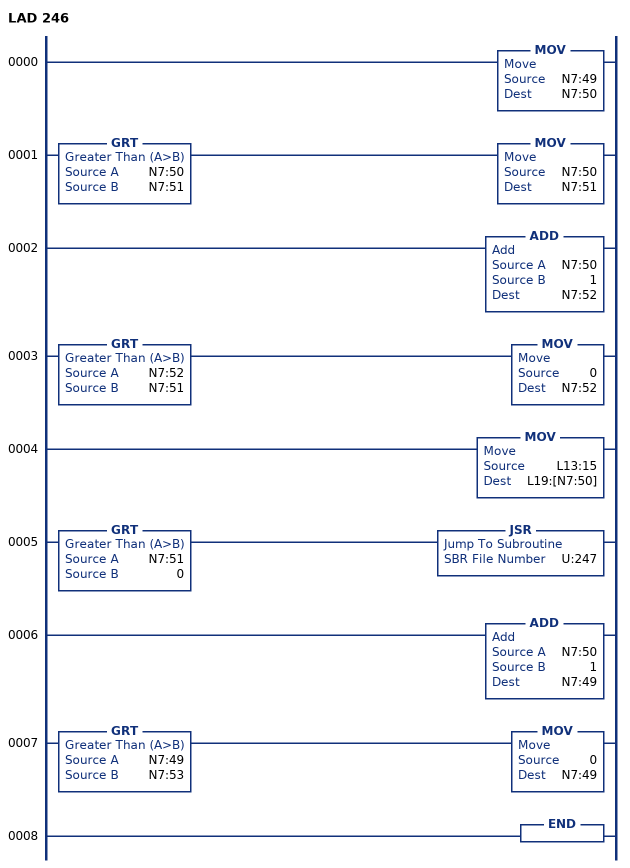
% Rung: 0 %
SOR MOV N7:49 N7:50 EOR
% Rung: 1 %
SOR GRT N7:50 N7:51 MOV N7:50 N7:51 EOR
% Rung: 2 %
SOR ADD N7:50 1 N7:52 EOR
% Rung: 3 %
SOR GRT N7:52 N7:51 MOV 0 N7:52 EOR
% Rung: 4 %
SOR MOV L13:15 L19:[N7:50] EOR
% Rung: 5 %
SOR GRT N7:51 0 JSR U:247 EOR
% Rung: 6 %
SOR ADD N7:50 1 N7:49 EOR
% Rung: 7 %
SOR GRT N7:49 N7:53 MOV 0 N7:49 EOR
% Rung: 8 %
SOR END EOR

LADDER 247
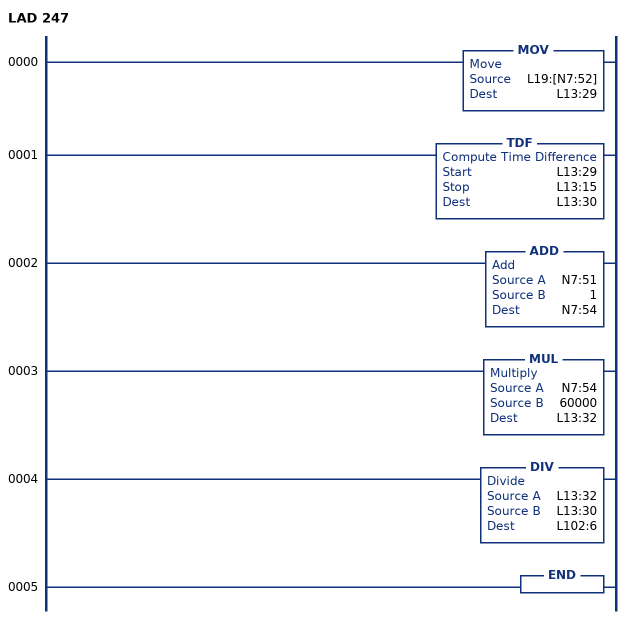
% Rung: 0 %
SOR MOV L19:[N7:52] L13:29 EOR
% Rung: 1 %
SOR TDF L13:29 L13:15 L13:30 EOR
% Rung: 2 %
SOR ADD N7:51 1 N7:54 EOR
% Rung: 3 %
SOR MUL N7:54 60000 L13:32 EOR
% Rung: 4 %
SOR DIV L13:32 L13:30 L102:6 EOR
% Rung: 5 %
SOR END EOR

LADDER 248
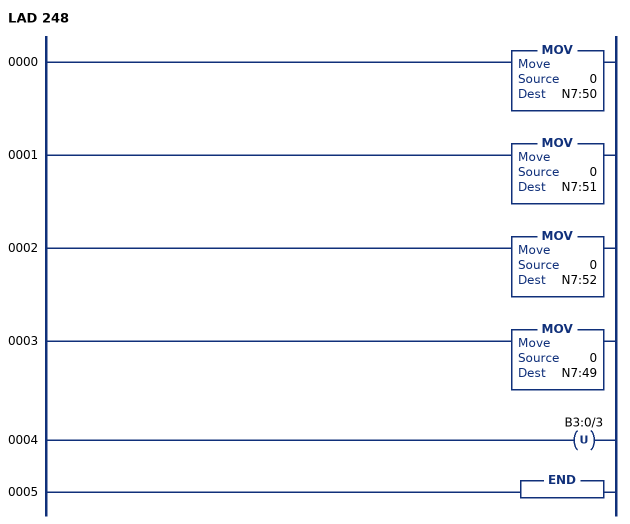
% Rung: 0 %
SOR MOV 0 N7:50 EOR
% Rung: 1 %
SOR MOV 0 N7:51 EOR
% Rung: 2 %
SOR MOV 0 N7:52 EOR
% Rung: 3 %
SOR MOV 0 N7:49 EOR
% Rung: 4 %
SOR OTU B3:0/3 EOR
% Rung: 5 %
SOR END EOR

LADDER 249
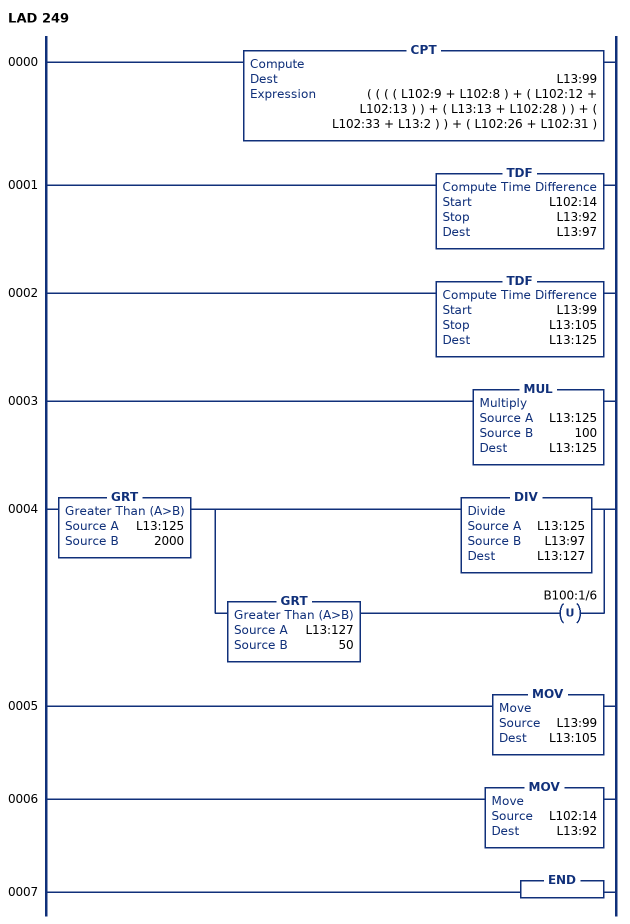
% Rung: 0 %
SOR CPT L13:99 " ( ( ( ( L102:9 + L102:8 ) + ( L102:12 + L102:13 ) ) + ( L13:13 + L102:28 ) ) + ( L102:33 + L13:2 ) ) + ( L102:26 + L102:31 ) " EOR
% Rung: 1 %
SOR TDF L102:14 L13:92 L13:97 EOR
% Rung: 2 %
SOR TDF L13:99 L13:105 L13:125 EOR
% Rung: 3 %
SOR MUL L13:125 100 L13:125 EOR
% Rung: 4 %
SOR GRT L13:125 2000 BST DIV L13:125 L13:97 L13:127 NXB GRT L13:127 50 OTU B100:1/6 BND EOR
% Rung: 5 %
SOR MOV L13:99 L13:105 EOR
% Rung: 6 %
SOR MOV L102:14 L13:92 EOR
% Rung: 7 %
SOR END EOR

LADDER 250
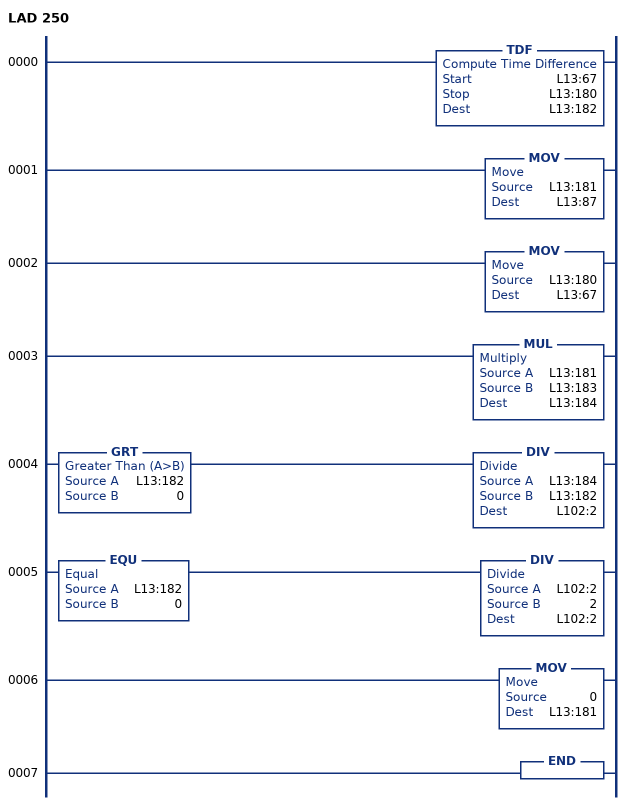
% Rung: 0 %
SOR TDF L13:67 L13:180 L13:182 EOR
% Rung: 1 %
SOR MOV L13:181 L13:87 EOR
% Rung: 2 %
SOR MOV L13:180 L13:67 EOR
% Rung: 3 %
SOR MUL L13:181 L13:183 L13:184 EOR
% Rung: 4 %
SOR GRT L13:182 0 DIV L13:184 L13:182 L102:2 EOR
% Rung: 5 %
SOR EQU L13:182 0 DIV L102:2 2 L102:2 EOR
% Rung: 6 %
SOR MOV 0 L13:181 EOR
% Rung: 7 %
SOR END EOR

LADDER 251
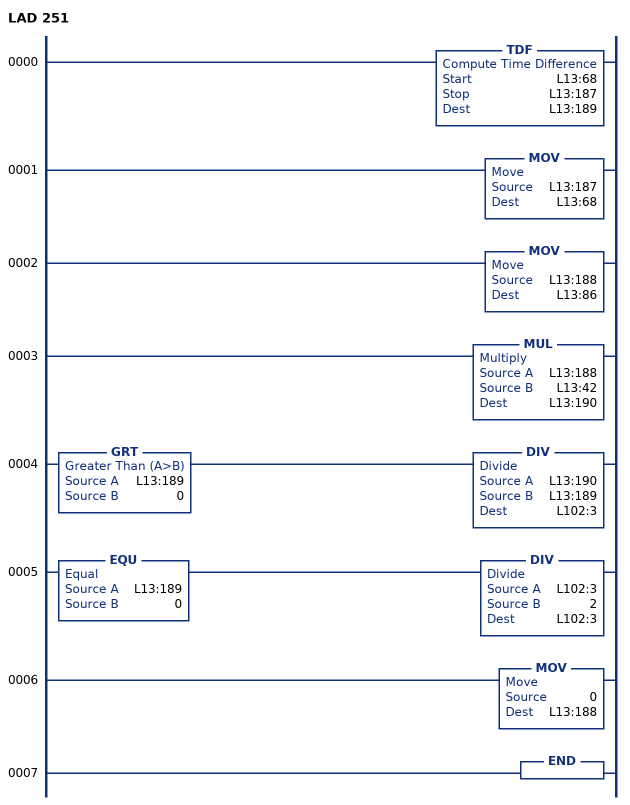
% Rung: 0 %
SOR TDF L13:68 L13:187 L13:189 EOR
% Rung: 1 %
SOR MOV L13:187 L13:68 EOR
% Rung: 2 %
SOR MOV L13:188 L13:86 EOR
% Rung: 3 %
SOR MUL L13:188 L13:42 L13:190 EOR
% Rung: 4 %
SOR GRT L13:189 0 DIV L13:190 L13:189 L102:3 EOR
% Rung: 5 %
SOR EQU L13:189 0 DIV L102:3 2 L102:3 EOR
% Rung: 6 %
SOR MOV 0 L13:188 EOR
% Rung: 7 %
SOR END EOR

LADDER 252
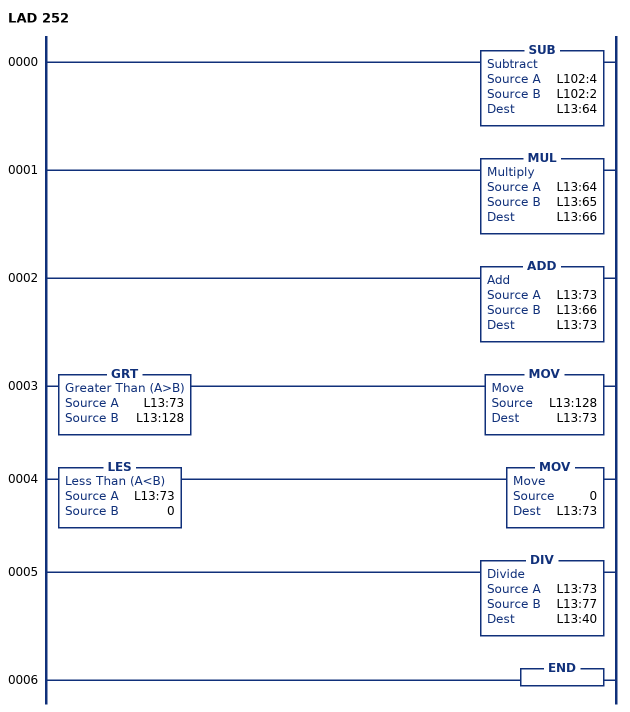
% Rung: 0 %
SOR SUB L102:4 L102:2 L13:64 EOR
% Rung: 1 %
SOR MUL L13:64 L13:65 L13:66 EOR
% Rung: 2 %
SOR ADD L13:73 L13:66 L13:73 EOR
% Rung: 3 %
SOR GRT L13:73 L13:128 MOV L13:128 L13:73 EOR
% Rung: 4 %
SOR LES L13:73 0 MOV 0 L13:73 EOR
% Rung: 5 %
SOR DIV L13:73 L13:77 L13:40 EOR
% Rung: 6 %
SOR END EOR

LADDER 253
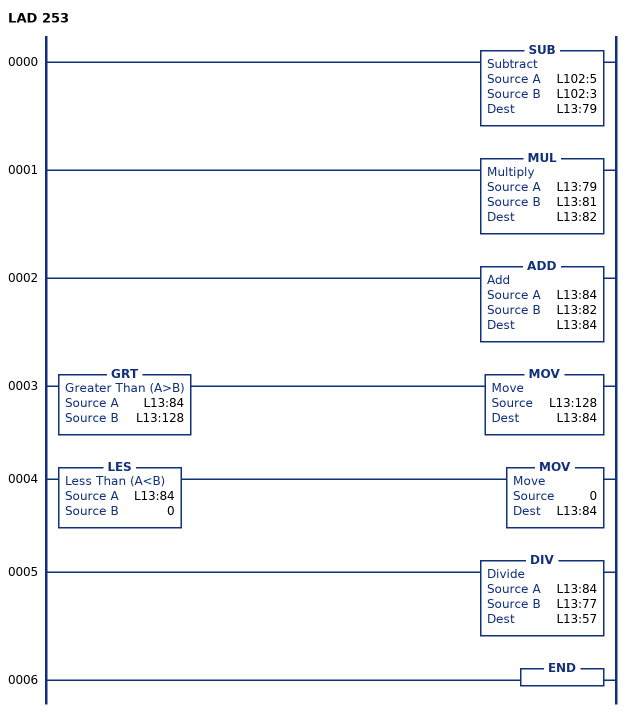
% Rung: 0 %
SOR SUB L102:5 L102:3 L13:79 EOR
% Rung: 1 %
SOR MUL L13:79 L13:81 L13:82 EOR
% Rung: 2 %
SOR ADD L13:84 L13:82 L13:84 EOR
% Rung: 3 %
SOR GRT L13:84 L13:128 MOV L13:128 L13:84 EOR
% Rung: 4 %
SOR LES L13:84 0 MOV 0 L13:84 EOR
% Rung: 5 %
SOR DIV L13:84 L13:77 L13:57 EOR
% Rung: 6 %
SOR END EOR

LADDER 254
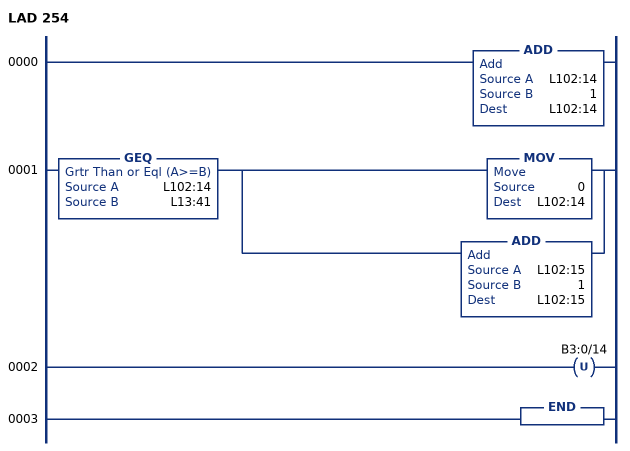
% Rung: 0 %
SOR ADD L102:14 1 L102:14 EOR
% Rung: 1 %
SOR GEQ L102:14 L13:41 BST MOV 0 L102:14 NXB ADD L102:15 1 L102:15 BND EOR
% Rung: 2 %
SOR OTU B3:0/14 EOR
% Rung: 3 %
SOR END EOR

LADDER 255
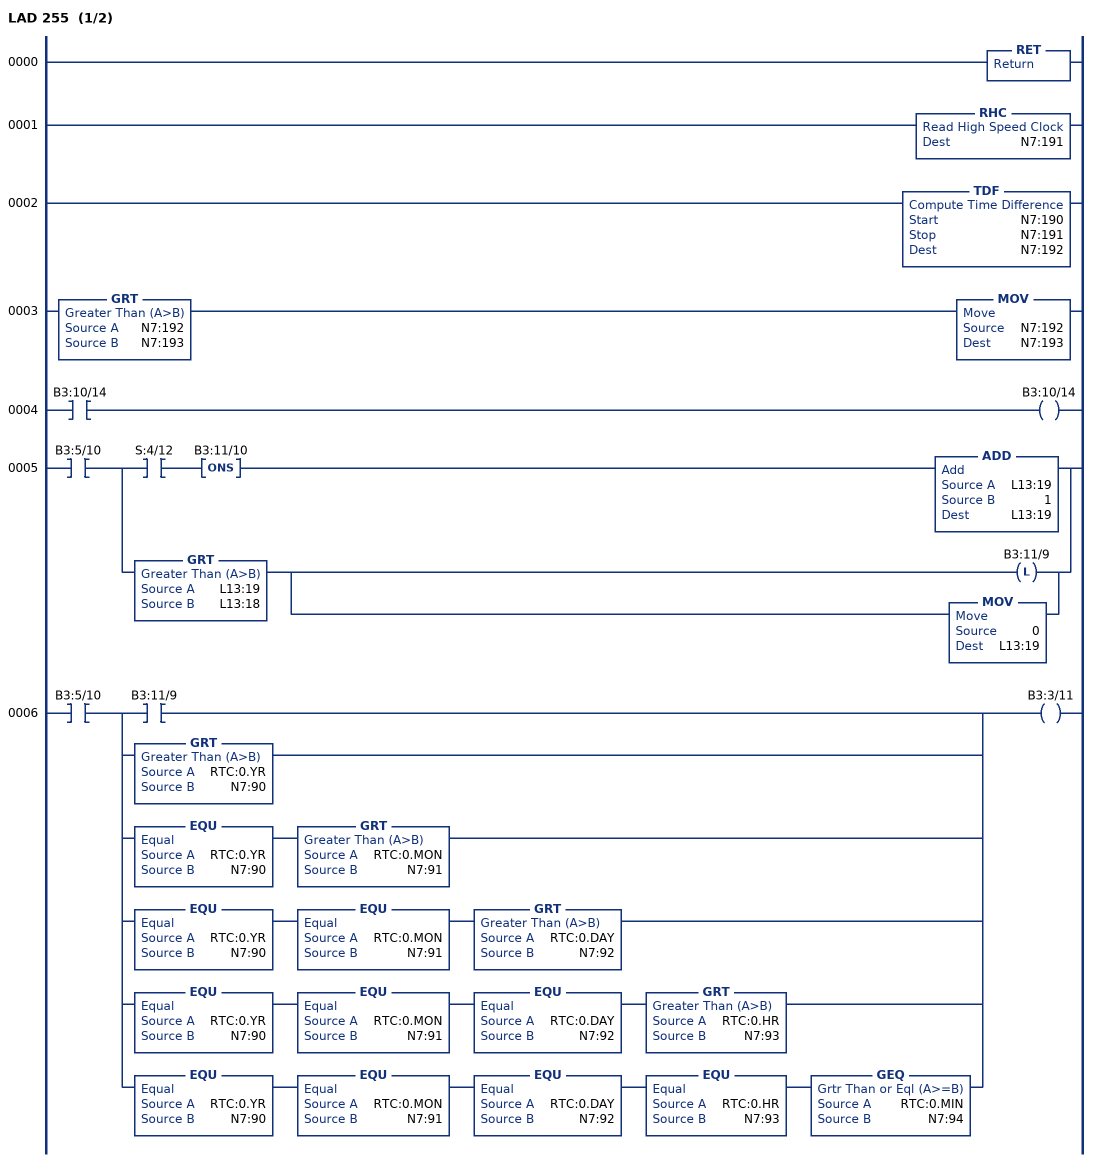
% Rung: 0 %
SOR RET EOR
% Rung: 1 %
SOR RHC N7:191 EOR
% Rung: 2 %
SOR TDF N7:190 N7:191 N7:192 EOR
% Rung: 3 %
SOR GRT N7:192 N7:193 MOV N7:192 N7:193 EOR
% Rung: 4 %
SOR XIC B3:10/14 OTE B3:10/14 EOR
% Rung: 5 %
SOR XIC B3:5/10 BST XIC S:4/12 ONS B3:11/10 ADD L13:19 1 L13:19 NXB GRT L13:19 L13:18 BST OTL B3:11/9 NXB MOV 0 L13:19 BND BND EOR
% Rung: 6 %
SOR XIC B3:5/10 BST XIC B3:11/9 NXB GRT RTC:0.YR N7:90 NXB EQU RTC:0.YR N7:90 GRT RTC:0.MON N7:91 NXB EQU RTC:0.YR N7:90 EQU RTC:0.MON N7:91 GRT RTC:0.DAY N7:92 NXB EQU RTC:0.YR N7:90 EQU RTC:0.MON N7:91 EQU RTC:0.DAY N7:92 GRT RTC:0.HR N7:93 NXB EQU RTC:0.YR N7:90 EQU RTC:0.MON N7:91 EQU RTC:0.DAY N7:92 EQU RTC:0.HR N7:93 GEQ RTC:0.MIN N7:94 BND OTE B3:3/11 EOR

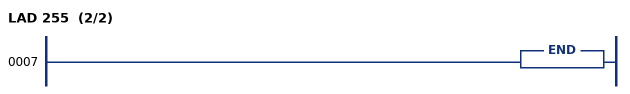
% Rung: 7 %
SOR END EOR

DATA TABLE (non-zero values as saved)
DATA B3
% B3:0 % 0X8830 0X0160 0X4001 0X5109 0X0EB3 0X0D34 0X0DB0 0X0421 0X2F80 0X22D0
% B3:10 % 0X21F4 0X000E 0X2000 0X0000 0X0000 0X0000 0X0000 0X0000 0X0000 0X0000
% B3:50 % 0X0001 0X0000 0X0000 0X0000 0X0000 0X0000 0X0000 0X0000 0X0000 0X0000
DATA T4
% .PRE .ACC %
% T4:0 % 0 2
% T4:1 % 150 0
% T4:2 % 400 0
% T4:3 % 500 76
% T4:4 % 1000 0
% T4:5 % 5 5
% T4:6 % 10 32766
% T4:7 % 666 0
% T4:8 % 20 7
% T4:9 % 50 7
% T4:10 % 200 200
% T4:11 % 111 0
% T4:12 % 40 42
% T4:13 % 250 0
% T4:14 % 666 0
% T4:15 % 1000 1002
% T4:16 % 400 0
% T4:17 % 100 59
% T4:18 % 5 0
% T4:19 % 300 0
% T4:20 % 200 0
% T4:21 % 200 0
% T4:22 % 200 0
% T4:23 % 250 0
% T4:24 % 666 0
% T4:25 % 666 0
% T4:26 % 666 0
% T4:27 % 250 0
% T4:28 % 250 0
% T4:29 % 5000 0
% T4:30 % 333 69
% T4:31 % 500 79
% T4:32 % 500 78
% T4:33 % 500 73
DATA C5
% .PRE .ACC %
% C5:0 % 32766 0
DATA R6
% .LEN .POS %
% R6:0 % 1250 0
% R6:1 % 1250 0
% R6:2 % 1050 0
% R6:3 % 1050 0
% R6:4 % 1250 0
% R6:5 % 1250 0
% R6:6 % 1713 0
% R6:7 % 1024 0
% R6:8 % 1024 0
% R6:9 % 3 0
% R6:10 % 2048 0
% R6:11 % 2048 0
% R6:12 % 10 0
% R6:13 % 10 0
% R6:14 % 10 0
% R6:15 % 10 0
% R6:16 % 1713 0
% R6:17 % 2048 0
% R6:18 % 2048 0
% R6:19 % 10 0
DATA N7
% N7:0 % 17247 3 1014 135 3 202 0 0 500 43
% N7:10 % 1000 0 0 2 20 20 1000 2000 50 1050
% N7:20 % 0 598 10 12 210 46 0 0 150 250
% N7:30 % 666 1453 150 0 17 1231 77 9 0 9
% N7:40 % 17 41 0 41 32767 1217 214 227 1636 6
% N7:50 % 5 16 6 16 17 1024 0 0 32766 0
% N7:60 % 1713 2048 2048 984 1034 1024 4999 5 400 400
% N7:70 % 100 200 300 400 90 190 290 390 13967 0
% N7:80 % 0 0 1239 1247 1247 1257 6 32 0 0
% N7:90 % 2011 4 4 12 1 6 32 222 222 12
% N7:100 % 1003 90 110 100 175 25 0 0 0 0
% N7:190 % 5698 17572 55 88 0 0 0 0 0 0
DATA F8
% F8:0 % 6
DATA L13
% L13:0 % 12165 115601 0 35109 182083
% L13:5 % 62 55 62 131362 55
% L13:10 % 58 6916237 30832 15 90
% L13:15 % 1605071481 -2147483648 2147483647 2147483647 82058
% L13:20 % 42216529 1963732491 777 33112 100
% L13:25 % 5304 2236 6399337 54 1257516236
% L13:30 % 347554360 62 1020000 1188692964 444
% L13:35 % 1 624336 0 0 0
% L13:40 % 12201 1000000000 1000000 1188692931 1532738498
% L13:45 % 1532738537 150 0 33 20590662
% L13:50 % 72333017 294744 1532738426 0 0
% L13:55 % 72332978 72333089 8943 -1783954998 -1783954972
% L13:60 % 26 104 -1783954986 600 -4
% L13:65 % 100 -400 -686583324 -686583191 12
% L13:70 % 1945503842 9 118 1220100 20590662
% L13:75 % 17067280 60 100 1532738435 -8
% L13:80 % 24 74 -592 7 894292
% L13:85 % 18228860 128 128 0 72333053
% L13:90 % 72333014 5 34844 5 1532738527
% L13:95 % 10 66272723 0 1532738561 92300
% L13:100 % 2147483647 6 1000 14 11717
% L13:105 % 92300 31 2099392 4691 2099386
% L13:110 % 6 100 50 1938587407 1945503621
% L13:115 % 1945503644 23 12 1945503632 26
% L13:120 % 4 3709 50 100 10
% L13:125 % 0 1945503842 2147483647 3276500 25145107
% L13:130 % 2 2 0 99 0
% L13:135 % 0 0 18228870 5 70
% L13:140 % 0 5 36 50 50
% L13:145 % 294745 5 5 5 9
% L13:150 % 12 20 516900 -516900 6916237
% L13:155 % 0 -10 0 0 4589052
% L13:160 % 7 29 24 1220 45
% L13:165 % 1945503860 1945503870 1945503860 1945503870 6706
% L13:170 % 12817 11770 11783 700 400
% L13:175 % 4 4 42 23 38
% L13:180 % -686526507 14 51246 1000000 128000000
% L13:185 % 1 0 -686526827 13 51147
% L13:190 % 128000000 0 0 0 0
DATA L19
% L19:0 % 1530305443 1530332613 1530429009 1532608863 1532722930
% L19:5 % 1532737645 1257516236 1257567107 1257591712 1257599369
% L19:10 % 1257607815 1257615308 1257623384 1257636706 1257643943
% L19:15 % 1257651424 1530296095 0 0 0
DATA L20
% L20:0 % 1530429861 1532609715 1532723785 1532725719 1532726224
% L20:5 % 1532726728 1532738498 1530199440 1530199944 1530200447
% L20:10 % 1530200952 1530201456 1530201960 1530202464 1530202969
% L20:15 % 1530203473 1530203978 1530204481 1530204984 1530205488
% L20:20 % 1530205991 1530206494 1530206998 1530207502 1530208006
% L20:25 % 1530208510 1530209015 1530209519 1530210023 1530210527
% L20:30 % 1530211030 1530211535 1530212039 1530212542 1530213046
% L20:35 % 1530213550 1530214055 1530214558 1530215062 1530215566
% L20:40 % 1530216071 1530216575 1530217080 1530217584 1530218088
% L20:45 % 1530218592 1530219095 1530296946 1530306295 1530333465
DATA L21
% L21:0 % 1944922040 1945471401 1945500151 1945500638 1945500766
% L21:5 % 1945500892 1945503860 1944885501 1944885501 1944885501
% L21:10 % 1944885501 1944885501 1944885501 1944885501 1944885501
% L21:15 % 1944885501 1944885501 1944885501 1944885501 1944885501
% L21:20 % 1944885501 1944885501 1944885501 1944885501 1944885501
% L21:25 % 1944885501 1944885501 1944885501 1944885501 1944885501
% L21:30 % 1944885501 1944885501 1944885501 1944885501 1944885501
% L21:35 % 1944885501 1944885501 1944885501 1944885501 1944885501
% L21:40 % 1944885501 1944885501 1944885501 1944885501 1944885501
% L21:45 % 1944885501 1944885501 1944888543 1944890899 1944897747
DATA L22
% L22:0 % 1257481069 1257490512 1257498604 1257509115 1257516794
% L22:5 % 1257567664 1257592269 1257599923 1257608372 1257615862
% L22:10 % 1257623940 1257637265 1257644499 1257651980 1283110057
% L22:15 % 1283110562 1283111067 1283111571 1290159732 1290160236
% L22:20 % 1290160741 1290161245 1290161749 1530296986 1530306334
% L22:25 % 1530333505 1530429901 1532609755 1532723824 1532725743
% L22:30 % 1532726250 1532726754 1532738537 1257111979 1257114467
% L22:35 % 1257128946 1257131427 1257152879 1257155369 1257160444
% L22:40 % 1257162927 1257191409 1257193891 1257205103 1257207593
% L22:45 % 1257400405 1257427688 1257445535 1257455613 1257463793
DATA L23
% L23:0 % 1942933757 1942937564 1942940828 1942945066 1942948162
% L23:5 % 1942968675 1942978596 1942981682 1942985089 1942988109
% L23:10 % 1942991367 1942996739 1942999655 1943002672 1944674498
% L23:15 % 1944674498 1944674498 1944674498 1944674498 1944674498
% L23:20 % 1944674498 1944674498 1944674498 1944888553 1944890909
% L23:25 % 1944897757 1944922050 1945471411 1945500161 1945500644
% L23:30 % 1945500772 1945500899 1945503870 1942784925 1942785928
% L23:35 % 1942791766 1942792767 1942801417 1942802421 1942804467
% L23:40 % 1942805468 1942816952 1942817953 1942822475 1942823478
% L23:45 % 1942901227 1942912230 1942919427 1942923491 1942926789
DATA L30
% L30:0 % 1097513510 1097513738 1097513967 1097514196 1097514426
% L30:5 % 1097514655 1097514883 1097515111 1097515339 1188692931
% L30:10 % 1071304952 1071305179 1071305406 1071305631 1071305859
% L30:15 % 1071306086 1071306312 1071306539 1071306765 1071306992
% L30:20 % 1071307217 1071307442 1071307668 1071307895 1071308121
% L30:25 % 1071308347 1071308573 1071308799 1071309024 1071309250
% L30:30 % 1071309476 1071429569 1071429795 1071431153 1071431379
% L30:35 % 1071431606 1088333039 1088333266 1088334623 1088334848
% L30:40 % 1088335075 1089808842 1089809070 1089810430 1089810657
% L30:45 % 1089810882 1092780028 1092791426 1092806921 1097513283
DATA L31
% L31:0 % 3522828 3522897 3522967 3523035 3523105
% L31:5 % 3523175 3523244 3523313 3523382 20590662
% L31:10 % 2077757 2077757 2077757 2077757 2077757
% L31:15 % 2077757 2077757 2077757 2077757 2077757
% L31:20 % 2077757 2077757 2077757 2077757 2077757
% L31:25 % 2077757 2077757 2077757 2077757 2077757
% L31:30 % 2077757 2077757 2077757 2077757 2077757
% L31:35 % 2077757 2077757 2077757 2077757 2077757
% L31:40 % 2077757 2077757 2077757 2077757 2077757
% L31:45 % 2077757 2091375 2094821 2099507 3522760
DATA L32
% L32:0 % 1530256824 1530257329 1530257832 1530258335 1530258840
% L32:5 % 1530259343 1530259847 1530260352 1530260857 1530261361
% L32:10 % 1530261865 1530262369 1530262873 1530263377 1530263881
% L32:15 % 1530264385 1530264889 1530265393 1530265898 1530266401
% L32:20 % 1530266906 1530267411 1530267914 1530268417 1530268923
% L32:25 % 1530269426 1530269930 1530270433 1530270936 1530271440
% L32:30 % 1530271943 1530296887 1530306235 1530333405 1530429801
% L32:35 % 1532609655 1532723710 1532725191 1532725697 1532726203
% L32:40 % 1532726709 1532738426 1530252792 1530253295 1530253800
% L32:45 % 1530254303 1530254807 1530255311 1530255815 1530256320
DATA L33
% L33:0 % 1944885501 1944885501 1944885501 1944885501 1944885501
% L33:5 % 1944885501 1944885501 1944885501 1944885501 1944885501
% L33:10 % 1944885501 1944885501 1944885501 1944885501 1944885501
% L33:15 % 1944885501 1944885501 1944885501 1944885501 1944885501
% L33:20 % 1944885501 1944885501 1944885501 1944885501 1944885501
% L33:25 % 1944885501 1944885501 1944885501 1944885501 1944885501
% L33:30 % 1944885501 1944888528 1944890884 1944897732 1944922025
% L33:35 % 1945471386 1945500132 1945500505 1945500633 1945500760
% L33:40 % 1945500887 1945503842 1944885501 1944885501 1944885501
% L33:45 % 1944885501 1944885501 1944885501 1944885501 1944885501
DATA B100
% B100:0 % 0X2780 0X18A8 0X0004 0X0000 0X0000 0X0000 0X0000 0X0000 0X0000 0X0000
DATA N101
% N101:0 % 118 0 0 0 1183 100 1002 1200 1212 1230
% N101:10 % 1240 1600 10 16383 1269 17365 3043 500 333 500
% N101:20 % 1000 500 400 0 0 0 500 500 0 0
DATA L102
% L102:0 % 40 10 2496 2498 2500
% L102:5 % 2500 0 21 0 0
% L102:10 % -516900 11 0 0 34844
% L102:15 % 0 30 10 30 10
% L102:20 % 11925 7 99017 0 29
% L102:25 % 33 0 91177564 81649 32
% L102:30 % 9 0 10 10636 0
% L102:35 % 174 302 0 999999 24
% L102:40 % 1 4 0 0 0
